// TIA Portal project "opc ua practice" (V16)

(* hardware
DEVICE "S71500/ET200MP station_1"  S7-1500 station
   slot 0: "Rail_0"  Rack  6ES7 590-1***0-0AA0
   slot 1: "server"  CPU 1516-3 PN/DP  6ES7 516-3AN01-0AB0  V2.8
      slot 3: "CPU display_1"  6ES7591-1BA00-0AA0
      slot 32768: "PROFINET interface_1"  X1
         slot 32769: "Port_1"  X1 P1
         slot 32770: "Port_2"  X1 P2
      slot 33024: "PROFINET interface_2"  X2
         slot 33025: "Port_1"  X2 P1
      slot 33280: "DP interface_1"  X3
      slot 34817: "Virtual CP interface port_1"  Virtual CP interface port  Virtual CP interface port
   slot 2: "AI 8xU/I/RTD/TC ST_1"  AI 8xU/I/RTD/TC ST  6ES7 531-7KF00-0AB0  V2.2
   slot 3: "DI 16x24VDC BA_1"  DI 16x24VDC BA  6ES7 521-1BH10-0AA0  V1.1
DEVICE "S71500/ET200MP station_2"  S7-1500 station
   slot 0: "Rail_0"  Rack  6ES7 590-1***0-0AA0
   slot 1: "client"  CPU 1516-3 PN/DP  6ES7 516-3AN01-0AB0  V2.8
      slot 3: "CPU display_1"  6ES7591-1BA00-0AA0
      slot 32768: "PROFINET interface_1"  X1
         slot 32769: "Port_1"  X1 P1
         slot 32770: "Port_2"  X1 P2
      slot 33024: "PROFINET interface_2"  X2
         slot 33025: "Port_1"  X2 P1
      slot 33280: "DP interface_1"  X3
      slot 34817: "Virtual CP interface port_1"  Virtual CP interface port  Virtual CP interface port
*)

// ===== PLC "server"  CPU 1516-3 PN/DP =====

VAR_GLOBAL   // PLC tag table "Default tag table"
   "start sms" AT %M0.0 : Bool;
   "stop sms" AT %M0.1 : Bool;
   "system on sms" AT %Q0.0 : Bool;
   "level meter sms" AT %ID0 : Real;
   "Tag_2" AT %MD4 : Real;
   "present level display sms" AT %QD34 : DInt;
   "set potentiometer sms" AT %ID4 : Real;
   "Tag_3" AT %MD8 : Real;
   "set level display sms" AT %QD38 : Real;
   "tag 13" AT %QD42 : DInt;
   "fill valve sms" AT %QD30 : Real;
   "reset" AT %Q0.1 : Bool;
   "start(1)" AT %I16.0 : Bool;
   "Discharge valve sms" AT %ID8 : Real;
   "Flow meter sms" AT %ID12 : Real;
END_VAR

DATA_BLOCK "db_server"   // DB1
{ S7_Optimized_Access := 'TRUE' }
VERSION : 0.1
   VAR
      motor_status : Bool;
      current : Int;
   END_VAR
BEGIN
END_DATA_BLOCK

ORGANIZATION_BLOCK "Main"   // OB1, LAD, ProgramCycle
TITLE = "Main Program Sweep (Cycle)"
{ S7_Optimized_Access := 'TRUE' }
VERSION : 0.1
   VAR_INPUT
      Initial_Call : Bool;   // Initial call of this OB
      Remanence : Bool;   // =True, if remanent data are available
   END_VAR
BEGIN

REGION Network 1
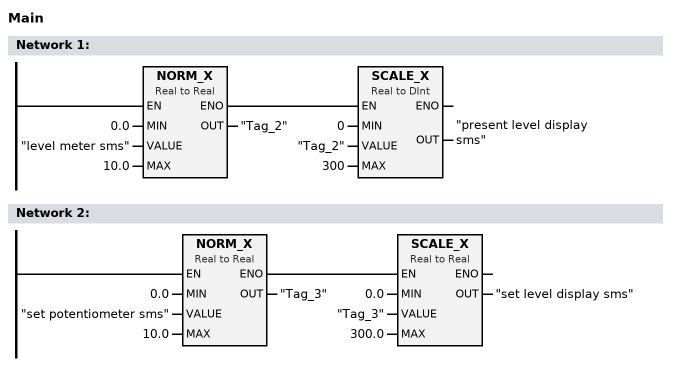
   RUNG wire#powerrail
      { S7_Templates := "[SrcType := Real, DestType := Real]" } Normalize(min := 0.0, value := "level meter sms", max := 10.0, out => "Tag_2")
      { S7_Templates := "[SrcType := Real, DestType := DInt]" } Scale(min := 0, value := "Tag_2", max := 300, out => "present level display sms")
   END_RUNG
   // the same network as SCL:
   "Tag_2" := NORM_X(MIN := 0.0, VALUE := "level meter sms", MAX := 10.0);
   "present level display sms" := SCALE_X(MIN := 0, VALUE := "Tag_2", MAX := 300);
END_REGION

REGION Network 2
   RUNG wire#powerrail
      { S7_Templates := "[SrcType := Real, DestType := Real]" } Normalize(min := 0.0, value := "set potentiometer sms", max := 10.0, out => "Tag_3")
      { S7_Templates := "[SrcType := Real, DestType := Real]" } Scale(min := 0.0, value := "Tag_3", max := 300.0, out => "set level display sms")
   END_RUNG
   // the same network as SCL:
   "Tag_3" := NORM_X(MIN := 0.0, VALUE := "set potentiometer sms", MAX := 10.0);
   "set level display sms" := SCALE_X(MIN := 0.0, VALUE := "Tag_3", MAX := 300.0);
END_REGION
END_ORGANIZATION_BLOCK

ORGANIZATION_BLOCK "Cyclic interrupt"   // OB30, LAD, CyclicInterrupt
{ S7_Optimized_Access := 'TRUE' }
VERSION : 0.1
   VAR_INPUT
      Initial_Call : Bool;   // Initial call of this OB
      Event_Count : Int;   // Events discarded
   END_VAR
BEGIN

REGION Network 1
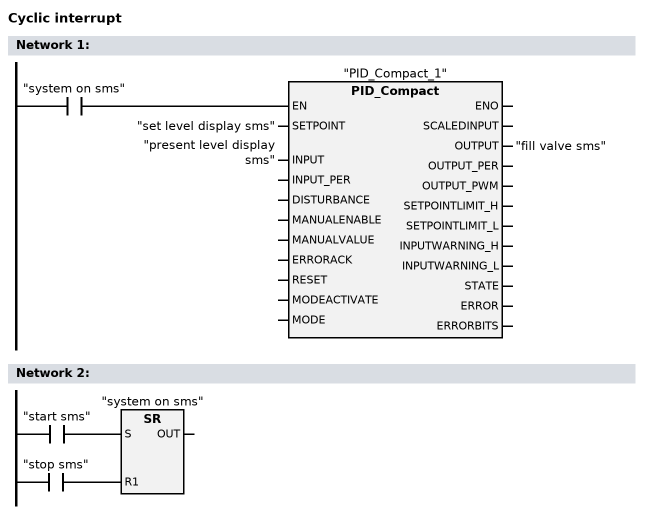
   IF "system on sms" THEN
       "PID_Compact_1"(Setpoint := "set level display sms",   // PID_Compact
                       Input := "present level display sms",
                       Output => "fill valve sms");
   END_IF;
END_REGION

REGION Network 2
   RUNG wire#powerrail
      Contact( "start sms" )
      S_SR(operand := "system on sms", r1 := wire#w1)
   END_RUNG
   RUNG wire#powerrail
      Contact( "stop sms" )
   END_RUNG wire#w1
   // the same network as SCL:
   IF "start sms" THEN
       "system on sms" := TRUE;   // SR flip-flop
   END_IF;
   IF "stop sms" THEN "system on sms" := FALSE; END_IF;
END_REGION
END_ORGANIZATION_BLOCK

// ===== PLC "client"  CPU 1516-3 PN/DP =====

DATA_BLOCK "Data_block_1"   // DB1
{ S7_Optimized_Access := 'TRUE' }
VERSION : 0.1
   VAR
      binary : Bool;
      analog : Int;
   END_VAR
BEGIN
END_DATA_BLOCK

ORGANIZATION_BLOCK "Main"   // OB1, LAD, ProgramCycle
TITLE = "Main Program Sweep (Cycle)"
{ S7_Optimized_Access := 'TRUE' }
VERSION : 0.1
   VAR_INPUT
      Initial_Call : Bool;   // Initial call of this OB
      Remanence : Bool;   // =True, if remanent data are available
   END_VAR
BEGIN
END_ORGANIZATION_BLOCK